KUKA KRL data list: KukaMatlabConnection_controller.dat

&ACCESS RVP
&REL 88
&PARAM TEMPLATE = C:\KRC\Roboter\Template\vorgabe
&PARAM EDITMASK = *
DEFDAT KukaMatlabConnection
;FOLD EXTERNAL DECLARATIONS;%{PE}%MKUKATPBASIS,%CEXT,%VCOMMON,%P
;FOLD BASISTECH EXT;%{PE}%MKUKATPBASIS,%CEXT,%VEXT,%P
EXT  BAS (BAS_COMMAND  :IN,REAL  :IN )
DECL INT SUCCESS
;ENDFOLD (BASISTECH EXT)
;FOLD USER EXT;%{E}%MKUKATPUSER,%CEXT,%VEXT,%P
;Make here your modifications

DECL RSIERR err
INT hEthernet,hmap
INT hDin,hDout1,hDout2,hDout3,hAxis,hPath,hMapDiO
INT UNIT_RSI
INT hAnaIn1,hAnaIn2,hAnaIn3,hAnaIn4,hAnaIn5,hAnaIn6,hAnaIn7
INT HP1,HP2
INT hsource

;ENDFOLD (USER EXT)
;ENDFOLD (EXTERNAL DECLERATIONS)
ENDDAT
